Universal Robots PolyScope program: TEST_SUB_105.urp

Program TEST_SUB_105 (installation=GD directory=/programs/GD createdIn=5.13.0 lastSavedIn=5.13.0 robotSerialNumber=20205000017)
Calibrated DH parameters: a=[-0.000157, -0.56303, -0.236706, -0.000074, -0.000109, 0]; d=[0.181705, 47.632387, 369.599619, -417.058513, 0.119878, 0.115667]; alpha=[1.570881, -0.005074, -0.001247, 1.56886, -1.570997, 0]; deltaTheta=[0, -0.405485, 5.544791, 1.143886, -0.000009, -0.000001]
InitVariablesNode
Robot Program (runOnlyOnce=true)
  var_2 := False
  SuppressedNode
    Force Frame feature=Bucket; selection=[1, 1, 1, 0, 0, 0]; wrench=[0, 0, 10, 0, 0, 0]; limitsForce=[0.01, 0.01, 0.015, 1.047198, 1.047198, 1.047198]; limitsMotion=[0.1, 0.1, 0.1, 0.349066, 0.349066, 0.349066]
      Wait Sleep waitTime=5
  var_3 := False
  ForceStartZ := CurrPos_p[2]
  Timer (action=Reset) variable(name=tm_cutoff)
  Timer (action=Start) variable=tm_cutoff
  Folder FORCE_CUTOFF
    Wait Sleep waitTime=0.02
    Script: zero_ftsensor()
    ForceStep := 0
    ForceFeature := Bucket
    ForceAxis := [1,1,1,0,0,0]
    ForceValue := [0.,0.,20.,0.,0.,0.]
    ForceType := 2
    CutOffZ := CutOffZ+CutOffZAdd
    CutOffZ := 0.1
    Loop While (checkContinuously=false) expression=tm_cutoff<GP_int_in[13]
      Switch expression=ForceStep
        Case (caseValue=0)
          ForceStep := 1
          IsBLLoad := False
          Timer (action=Reset) variable(name=tm_blload)
          ForceLimit := [0.01,0.01,0.015,d2r(10.),d2r(10.),d2r(10.)]
          Script: force_mode(Bucket,ForceAxis,ForceValue,ForceType,ForceLimit)
        Case (caseValue=1)
          If var_2 and ( not IsBLLoad) (checkContinuously=true)
            IsBLLoad := True
            Timer (action=Reset) variable=tm_blload
            Timer (action=Start) variable=tm_blload
          ElseIf ( not var_2) and IsBLLoad
            IsBLLoad := False
            Timer (action=Stop) variable=tm_blload
          ElseIf var_2 and IsBLLoad
            If tm_blload>TM_BLLoad
              IsBLLoad := False
              Timer (action=Stop) variable=tm_blload
              ForceStep := 2
              ForceLimit := [0.01,0.01,0.25,d2r(10.),d2r(10.),d2r(10.)]
              Script: force_mode(Bucket,ForceAxis,ForceValue,ForceType,ForceLimit)
          Else 
            var_1 := tm_cutoff
            If tm_cutoff>1
              var_2 := True
        Case (caseValue=2)
          If CurrPos_p[2]>ForceStartZ+CutOffZ
            ForceStep := 3
            Script: break
          If var_3 and ( not IsBLLoad)
            IsBLLoad := True
            Timer (action=Reset) variable=tm_blload
            Timer (action=Start) variable=tm_blload
          ElseIf ( not var_3) and IsBLLoad
            IsBLLoad := False
            Timer (action=Stop) variable=tm_blload
          ElseIf var_3 and IsBLLoad
            If tm_blload>TM_BLLoad
              IsBLLoad := False
              Timer (action=Stop) variable=tm_blload
              Script: break
      Script: sync()
    Script: end_force_mode()
  Timer (action=Stop) variable=tm_cutoff
  Popup Message (haltProgram=false inputType=Variable) variable=ForceStep
Thread スレッド_1 (runOnlyOnce=false)
  Script: CurrPos_p=get_actual_tcp_pose()
